SUBAPPLICATION Uebung_041_AX (* Lauflicht 8 mit einer Taste, mit Plug and Socket *)
  (* Standard: 61499-2; Description: Copyright (c) 2026 Meisterschulen am Ostbahnhof This program and the accompanying materials are made available under the terms of the Eclipse Public License 2.0 which is available at https://www.eclipse.org/legal/epl-2.0/ SPDX-License-Identifier: EPL-2.0 *)
  (* Version 1.0, 2026-09-09, Franz Höpfinger, Meisterschulen am Ostbahnhof, initial API and implementation and/or initial documentation *)
  PACKAGE Uebungen;
  IMPORT Uebungen::const::UT::DefaultPool::OutputNumber_N1;
  IMPORT logiBUS::io::DI::logiBUS_DI::Input_I1;
  IMPORT logiBUS::io::DI::logiBUS_DI::Input_I2;
  IMPORT logiBUS::io::DI::logiBUS_DI::Input_I4;
  IMPORT logiBUS::io::DI::logiBUS_DI_Events::BUTTON_SINGLE_CLICK;
  IMPORT logiBUS::io::DQ::logiBUS_DO::Output_Q1;
  IMPORT logiBUS::io::DQ::logiBUS_DO::Output_Q2;
  IMPORT logiBUS::io::DQ::logiBUS_DO::Output_Q3;
  IMPORT logiBUS::io::DQ::logiBUS_DO::Output_Q4;
  IMPORT logiBUS::io::DQ::logiBUS_DO::Output_Q5;
  IMPORT logiBUS::io::DQ::logiBUS_DO::Output_Q6;
  IMPORT logiBUS::io::DQ::logiBUS_DO::Output_Q7;
  IMPORT logiBUS::io::DQ::logiBUS_DO::Output_Q8;
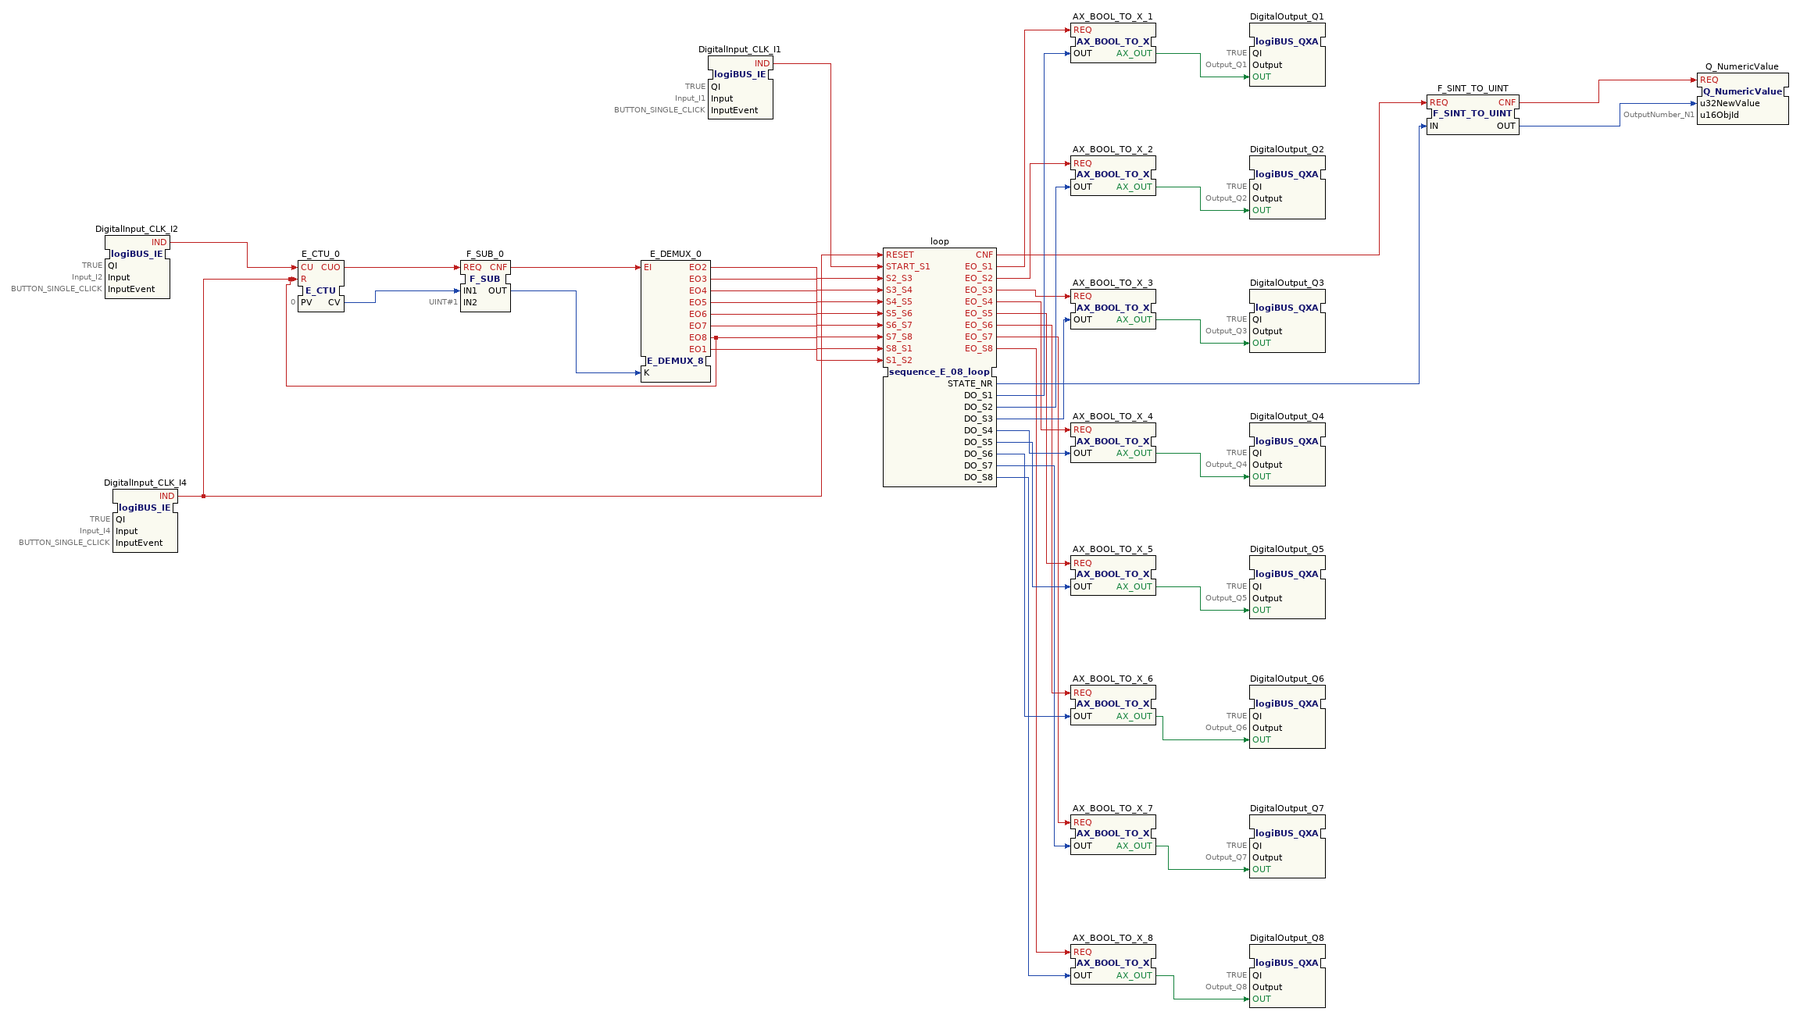
  FBS
    DigitalOutput_Q1 : logiBUS::io::DQ::logiBUS_QXA(QI := TRUE, Output := Output_Q1);
    DigitalOutput_Q2 : logiBUS::io::DQ::logiBUS_QXA(QI := TRUE, Output := Output_Q2);
    DigitalOutput_Q3 : logiBUS::io::DQ::logiBUS_QXA(QI := TRUE, Output := Output_Q3);
    DigitalOutput_Q4 : logiBUS::io::DQ::logiBUS_QXA(QI := TRUE, Output := Output_Q4);
    DigitalInput_CLK_I1 : logiBUS::io::DI::logiBUS_IE(QI := TRUE, Input := Input_I1, InputEvent := BUTTON_SINGLE_CLICK);
    DigitalInput_CLK_I4 : logiBUS::io::DI::logiBUS_IE(QI := TRUE, Input := Input_I4, InputEvent := BUTTON_SINGLE_CLICK);
    DigitalOutput_Q5 : logiBUS::io::DQ::logiBUS_QXA(QI := TRUE, Output := Output_Q5);
    DigitalOutput_Q6 : logiBUS::io::DQ::logiBUS_QXA(QI := TRUE, Output := Output_Q6);
    DigitalOutput_Q7 : logiBUS::io::DQ::logiBUS_QXA(QI := TRUE, Output := Output_Q7);
    DigitalOutput_Q8 : logiBUS::io::DQ::logiBUS_QXA(QI := TRUE, Output := Output_Q8);
    Q_NumericValue : isobus::UT::Q::Q_NumericValue(u16ObjId := OutputNumber_N1);
    F_SINT_TO_UINT : iec61131::conversion::F_SINT_TO_UINT;
    loop : logiBUS::utils::sequence::event::sequence_E_08_loop;
    E_CTU_0 : iec61499::events::E_CTU(PV := 0);
    DigitalInput_CLK_I2 : logiBUS::io::DI::logiBUS_IE(QI := TRUE, Input := Input_I2, InputEvent := BUTTON_SINGLE_CLICK);
    F_SUB_0 : iec61131::arithmetic::F_SUB(IN2 := UINT#1);
    E_DEMUX_0 : iec61499::events::E_DEMUX_8;
    AX_BOOL_TO_X_1 : adapter::conversion::unidirectional::AX_BOOL_TO_X;
    AX_BOOL_TO_X_2 : adapter::conversion::unidirectional::AX_BOOL_TO_X;
    AX_BOOL_TO_X_3 : adapter::conversion::unidirectional::AX_BOOL_TO_X;
    AX_BOOL_TO_X_4 : adapter::conversion::unidirectional::AX_BOOL_TO_X;
    AX_BOOL_TO_X_5 : adapter::conversion::unidirectional::AX_BOOL_TO_X;
    AX_BOOL_TO_X_6 : adapter::conversion::unidirectional::AX_BOOL_TO_X;
    AX_BOOL_TO_X_7 : adapter::conversion::unidirectional::AX_BOOL_TO_X;
    AX_BOOL_TO_X_8 : adapter::conversion::unidirectional::AX_BOOL_TO_X;
  END_FBS
  EVENT_CONNECTIONS
    F_SINT_TO_UINT.CNF TO Q_NumericValue.REQ;
    DigitalInput_CLK_I4.IND TO loop.RESET;
    loop.CNF TO F_SINT_TO_UINT.REQ;
    loop.EO_S1 TO AX_BOOL_TO_X_1.REQ;
    loop.EO_S2 TO AX_BOOL_TO_X_2.REQ;
    loop.EO_S3 TO AX_BOOL_TO_X_3.REQ;
    loop.EO_S4 TO AX_BOOL_TO_X_4.REQ;
    loop.EO_S5 TO AX_BOOL_TO_X_5.REQ;
    loop.EO_S6 TO AX_BOOL_TO_X_6.REQ;
    loop.EO_S7 TO AX_BOOL_TO_X_7.REQ;
    loop.EO_S8 TO AX_BOOL_TO_X_8.REQ;
    DigitalInput_CLK_I1.IND TO loop.START_S1;
    DigitalInput_CLK_I2.IND TO E_CTU_0.CU;
    E_CTU_0.CUO TO F_SUB_0.REQ;
    DigitalInput_CLK_I4.IND TO E_CTU_0.R;
    F_SUB_0.CNF TO E_DEMUX_0.EI;
    E_DEMUX_0.EO2 TO loop.S2_S3;
    E_DEMUX_0.EO3 TO loop.S3_S4;
    E_DEMUX_0.EO4 TO loop.S4_S5;
    E_DEMUX_0.EO5 TO loop.S5_S6;
    E_DEMUX_0.EO6 TO loop.S6_S7;
    E_DEMUX_0.EO7 TO loop.S7_S8;
    E_DEMUX_0.EO8 TO loop.S8_S1;
    E_DEMUX_0.EO8 TO E_CTU_0.R;
    E_DEMUX_0.EO1 TO loop.S1_S2;
  END_CONNECTIONS
  DATA_CONNECTIONS
    F_SINT_TO_UINT.OUT TO Q_NumericValue.u32NewValue;
    loop.STATE_NR TO F_SINT_TO_UINT.IN;
    loop.DO_S1 TO AX_BOOL_TO_X_1.OUT;
    loop.DO_S2 TO AX_BOOL_TO_X_2.OUT;
    loop.DO_S3 TO AX_BOOL_TO_X_3.OUT;
    loop.DO_S4 TO AX_BOOL_TO_X_4.OUT;
    loop.DO_S5 TO AX_BOOL_TO_X_5.OUT;
    loop.DO_S6 TO AX_BOOL_TO_X_6.OUT;
    loop.DO_S7 TO AX_BOOL_TO_X_7.OUT;
    loop.DO_S8 TO AX_BOOL_TO_X_8.OUT;
    E_CTU_0.CV TO F_SUB_0.IN1;
    F_SUB_0.OUT TO E_DEMUX_0.K;
  END_CONNECTIONS
  ADAPTER_CONNECTIONS
    AX_BOOL_TO_X_1.AX_OUT TO DigitalOutput_Q1.OUT;
    AX_BOOL_TO_X_2.AX_OUT TO DigitalOutput_Q2.OUT;
    AX_BOOL_TO_X_3.AX_OUT TO DigitalOutput_Q3.OUT;
    AX_BOOL_TO_X_4.AX_OUT TO DigitalOutput_Q4.OUT;
    AX_BOOL_TO_X_5.AX_OUT TO DigitalOutput_Q5.OUT;
    AX_BOOL_TO_X_6.AX_OUT TO DigitalOutput_Q6.OUT;
    AX_BOOL_TO_X_7.AX_OUT TO DigitalOutput_Q7.OUT;
    AX_BOOL_TO_X_8.AX_OUT TO DigitalOutput_Q8.OUT;
  END_CONNECTIONS
END_SUBAPPLICATION
